{attribute 'GeneratedUsingTerminal: EK1122-0000-0018'}
{attribute addProperty BoxType "EK1122-0000-0018"}
{attribute addProperty Id "R8_AB0_EPP1322_0001R8_AB0_EPP1322_0001_1BB6BCA8290"}
{attribute addProperty CRC "3880536930"}
{attribute addProperty Size "290"}
{attribute addProperty Name "R8_A2 (EK1122)"}
TYPE R8_A2_EK1122_E74C4B62 EXTENDS EK1122_1FC0878B :
STRUCT
	{attribute addProperty Name "R8_AB0 (EPP1322-0001)"}
	{attribute addProperty PreviousPort "R8_A2 (EK1122) : D"}
	{attribute addProperty SyncUnit "default"}
	R8_AB0_EPP1322_0001 : R8_AB0_EPP1322_0001_1BB6BCA8;
END_STRUCT
END_TYPE

(* stored: Version 1.2.0.0, ProductVersion 3.1.4024.11
   DUT R8_A2_EK1122_E74C4B62: Id {675a43ef-8bb0-0ddf-187b-2a678f0fa13e} *)
